PROGRAM Q3
VAR
	// INT : num1 := 1;
	// DataType and VarName are wrong way round
	num1 : INT := 1;
END_VAR

END_PROGRAM

(* stored: Version 1.1.0.1, ProductVersion 3.1.4024.12
   POU Q3: Id {fa57265e-fa60-475b-8b69-c379cbc68b91}, SpecialFunc None *)
